// Mitsubishi GX Works2 project: GROUP13   PLC: FX3G

// global labels: Global1
VAR_GLOBAL
  M_StartBlinking AT M100 : BOOL;
  light_generator AT M101 : BOOL;
  TC_BLINK_1 AT TC1 : BOOL;
END_VAR
VAR_GLOBAL CONSTANT
  CONSTANT3_word : INT := 3;
END_VAR
VAR_GLOBAL
  TC_BLINK_2 AT TC2 : BOOL;
  TS_BLINK_1 AT TS1 : BOOL;
  TS_BLINK_2 AT TS2 : BOOL;
  M_BLINKING_LIGHT1 AT M201 : BOOL;
  M_BLINKING_LIGHT2 AT M202 : BOOL;
  Sw_1_Collect AT X001 : BOOL;
  Sw_2_Wash AT X002 : BOOL;
  Sw_3_QA AT X003 : BOOL;
  Sw4 AT X004 : BOOL;
  Sw5 AT X005 : BOOL;
  Sw6 AT X006 : BOOL;
  Sw_7_Emergency AT X007 : BOOL;
  Sw_10_StartDay AT X010 : BOOL;
  Sw_11_Squeeze AT X011 : BOOL;
  Li_1_Collected AT Y001 : BOOL;
  Li_2_Squeeze AT Y002 : BOOL;
  Li_3_Squeeze AT Y003 : BOOL;
  Li_4_QA_Succsed AT Y004 : BOOL;
  Li_5_Wash AT Y005 : BOOL;
  Li6 AT Y006 : BOOL;
  Li7 AT Y007 : BOOL;
  Li_10_Day AT Y010 : BOOL;
  Li11 AT Y011 : BOOL;
  CC_Start_Squeeze_0 AT CC0 : BOOL;
  CS_Start_Squeeze_0 AT CS0 : BOOL;
  TC_Squeeze_10 AT TC10 : BOOL;
END_VAR
VAR_GLOBAL CONSTANT
  CONSTANT2_word : INT := 2;
  CONSTANT30_word : INT := 30;
END_VAR
VAR_GLOBAL
  TS_Squeeze_10 AT TS10 : BOOL;
END_VAR
VAR_GLOBAL CONSTANT
  CONSTANT1_float : REAL := 1;
END_VAR
VAR_GLOBAL
  REG_InvetoryOrange AT D1100 : REAL;
  REG_InvetoryClementine AT D1102 : REAL;
  REG_InvetoryPomelo AT D1104 : REAL;
END_VAR
VAR_GLOBAL CONSTANT
  CONSTANT2_float : REAL := 2;
END_VAR
VAR_GLOBAL
  M_canStartDay AT M0 : BOOL;
  M_TurnOffAll AT M10 : BOOL;
END_VAR
VAR_GLOBAL CONSTANT
  CONSTANT0_float : REAL;
END_VAR
VAR_GLOBAL
  REG_Squeeze AT D1112 : REAL;
  REG_Juice AT D1114 : REAL;
  REG_Storage AT D1116 : REAL;
  TC_CloseDayTimer_3 AT TC3 : BOOL;
  TS_CloseDayTimer_3 AT TS3 : BOOL;
END_VAR
VAR_GLOBAL CONSTANT
  CONSTANT1_word : INT := 1;
END_VAR
VAR_GLOBAL
  M_StartWash AT M1 : BOOL;
  TC_Wash_0 AT TC0 : BOOL;
  TS_Wash_0 AT TS0 : BOOL;
END_VAR
VAR_GLOBAL CONSTANT
  CONSTANT_maxOrange : REAL := 100;
END_VAR
VAR_GLOBAL
  REG_TempWashOrange AT D1118 : REAL;
  M_checkMinimum AT M3 : BOOL;
  REG_minimumPC AT D1120 : REAL;
  M_proportionAdjusment AT M8 : BOOL;
  M_foundMinimum AT M4 : BOOL;
  REG_MinimumPOC AT D1126 : REAL;
  REG_WashOrange AT D1106 : REAL;
  REG_WashClementine AT D1108 : REAL;
  REG_WashPomelo AT D1110 : REAL;
  M_OinWash AT M5 : BOOL;
  M_PinWash AT M6 : BOOL;
  M_CinWash AT M7 : BOOL;
  REG_HalfMinimumPOC AT D1122 : REAL;
  M_Check_QA_1 AT M11 : BOOL;
  M_Check_QA_2 AT M12 : BOOL;
  M_QA_PASSED AT M15 : BOOL;
  M_STARTQA AT M13 : BOOL;
  QA_COUNTER AT CC3 : BOOL;
  CS_MAX_QA AT CS3 : BOOL;
  SW_Analog2_QA AT D8281 : INT;
  REG_QA_value AT D1150 : INT;
END_VAR
VAR_GLOBAL CONSTANT
  CONSTANT5_word : INT := 5;
END_VAR
VAR_GLOBAL
  TC_QA_TEST_PASSED AT TC201 : BOOL;
END_VAR
VAR_GLOBAL CONSTANT
  CONSTANT500_word : INT := 500;
END_VAR
VAR_GLOBAL
  TS_QA_TEST_PASSED AT TS201 : BOOL;
  M_InvetoryOrange_21 AT M21 : BOOL;
  M_InvetoryPomelo_22 AT M22 : BOOL;
  M_InvetoryClementine_20 AT M20 : BOOL;
  M_NotInWash AT M23 : BOOL;
  M_NotInSqueze AT M24 : BOOL;
  M_NotInJuice AT M25 : BOOL;
  REG_keg AT D1128 : INT;
END_VAR
VAR_GLOBAL CONSTANT
  CONSTANT_15_word : INT := 15;
END_VAR
VAR_GLOBAL
  analog_output AT D8282 : INT;
  M_KegNumberFound AT M36 : BOOL;
  REG_keg_FLOAT AT D1132 : REAL;
END_VAR
VAR_GLOBAL CONSTANT
  CONSTANT50_float : REAL := 50;
END_VAR
VAR_GLOBAL
  TS_SHIPMENT_5 AT TS5 : BOOL;
  TC_shipment_5 AT TC5 : BOOL;
  M_SHIMPMENTOVER15 AT M33 : BOOL;
  TC_Shipment_4 AT TC4 : BOOL;
  TS_SHIPMENT_4 AT TS4 : BOOL;
END_VAR
VAR_GLOBAL CONSTANT
  CONSTANT382_1inanalog : INT := 382;
  CONSTANT2020_5inanalog : INT := 2020;
  CONSTANT80_float : REAL := 80;
  CONSTANT_400_word : INT := 400;
END_VAR

// task Task_01 (event TRUE, interval 0, priority 31): POU_01

PROGRAM POU_01
(* structured ladder/FBD written out as ST: instructions are called as NAME(EN, inputs, outputs); _pN, _eN, _tN stand for wires *)
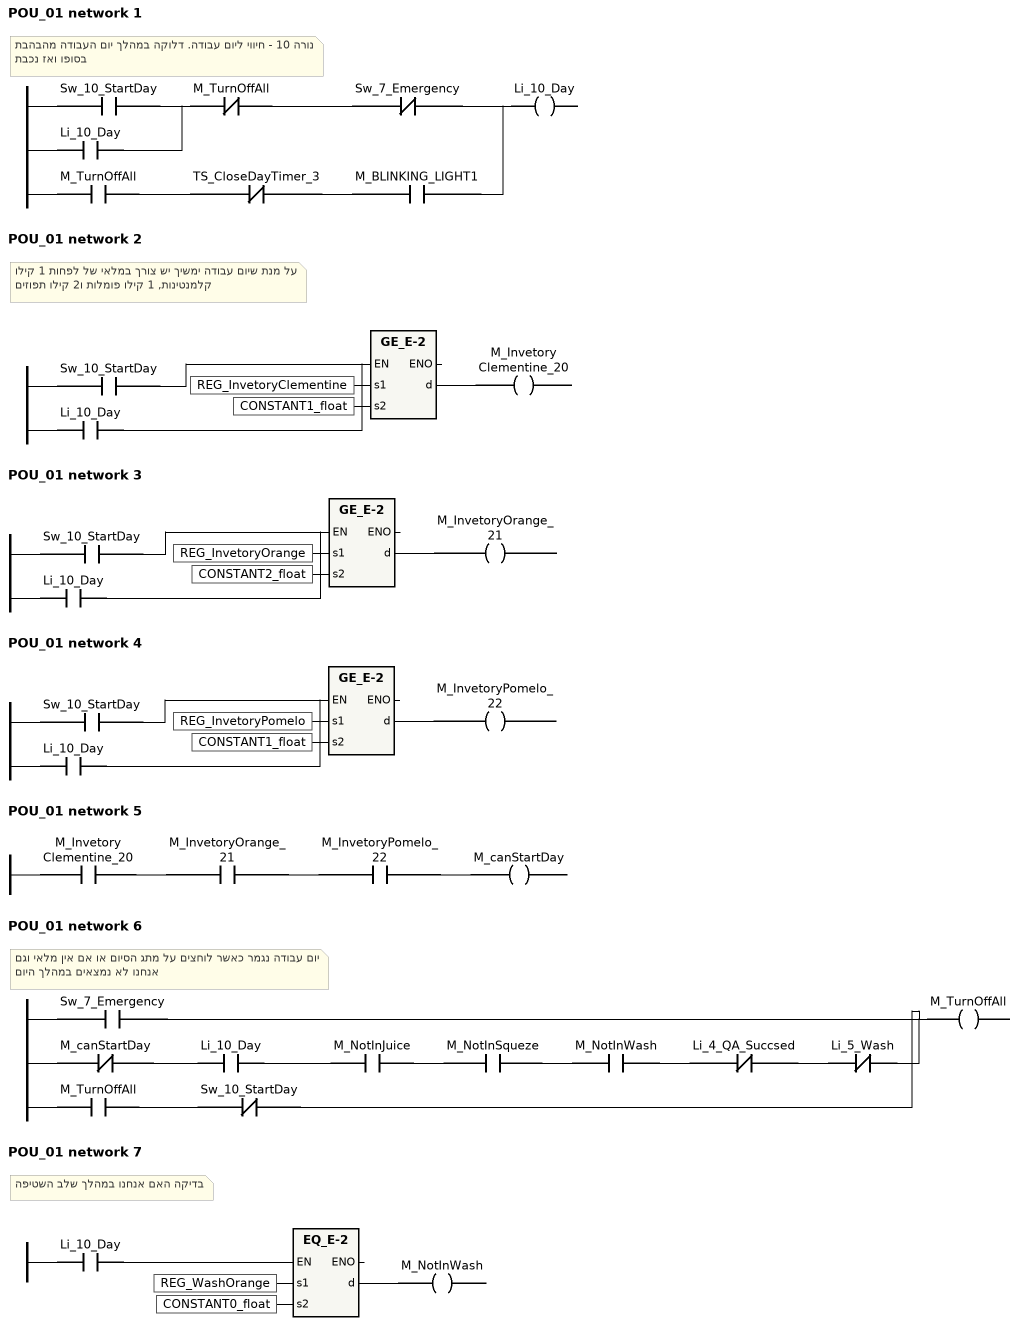
(* network 1 *)
(* נורה 10 - חיווי ליום עבודה. דלוקה במהלך יום העבודה מהבהבת בסופו ואז נכבת *)
Li_10_Day := (((Sw_10_StartDay OR Li_10_Day) AND NOT M_TurnOffAll) AND NOT Sw_7_Emergency) OR (M_TurnOffAll AND NOT TS_CloseDayTimer_3 AND M_BLINKING_LIGHT1);
(* network 2 *)
(* על מנת שיום עבודה ימשיך יש צורך במלאי של לפחות 1 קילו קלמנטינות, 1 קילו פומלות ו2 קילו תפוזים *)
GE_E(Sw_10_StartDay OR Li_10_Day, REG_InvetoryClementine, CONSTANT1_float, _t1);
M_InvetoryClementine_20 := _t1;
(* network 3 *)
GE_E(Sw_10_StartDay OR Li_10_Day, REG_InvetoryOrange, CONSTANT2_float, _t1);
M_InvetoryOrange_21 := _t1;
(* network 4 *)
GE_E(Sw_10_StartDay OR Li_10_Day, REG_InvetoryPomelo, CONSTANT1_float, _t1);
M_InvetoryPomelo_22 := _t1;
(* network 5 *)
M_canStartDay := M_InvetoryClementine_20 AND M_InvetoryOrange_21 AND M_InvetoryPomelo_22;
(* network 6 *)
(* יום עבודה נגמר כאשר לוחצים על מתג הסיום או אם אין מלאי וגם אנחנו לא נמצאים במהלך היום *)
M_TurnOffAll := Sw_7_Emergency OR (NOT M_canStartDay AND Li_10_Day AND M_NotInJuice AND M_NotInSqueze AND M_NotInWash AND NOT Li_4_QA_Succsed AND NOT Li_5_Wash) OR (M_TurnOffAll AND NOT Sw_10_StartDay);
(* network 7 *)
(* בדיקה האם אנחנו במהלך שלב השטיפה *)
EQ_E(Li_10_Day, REG_WashOrange, CONSTANT0_float, _t1);
M_NotInWash := _t1;
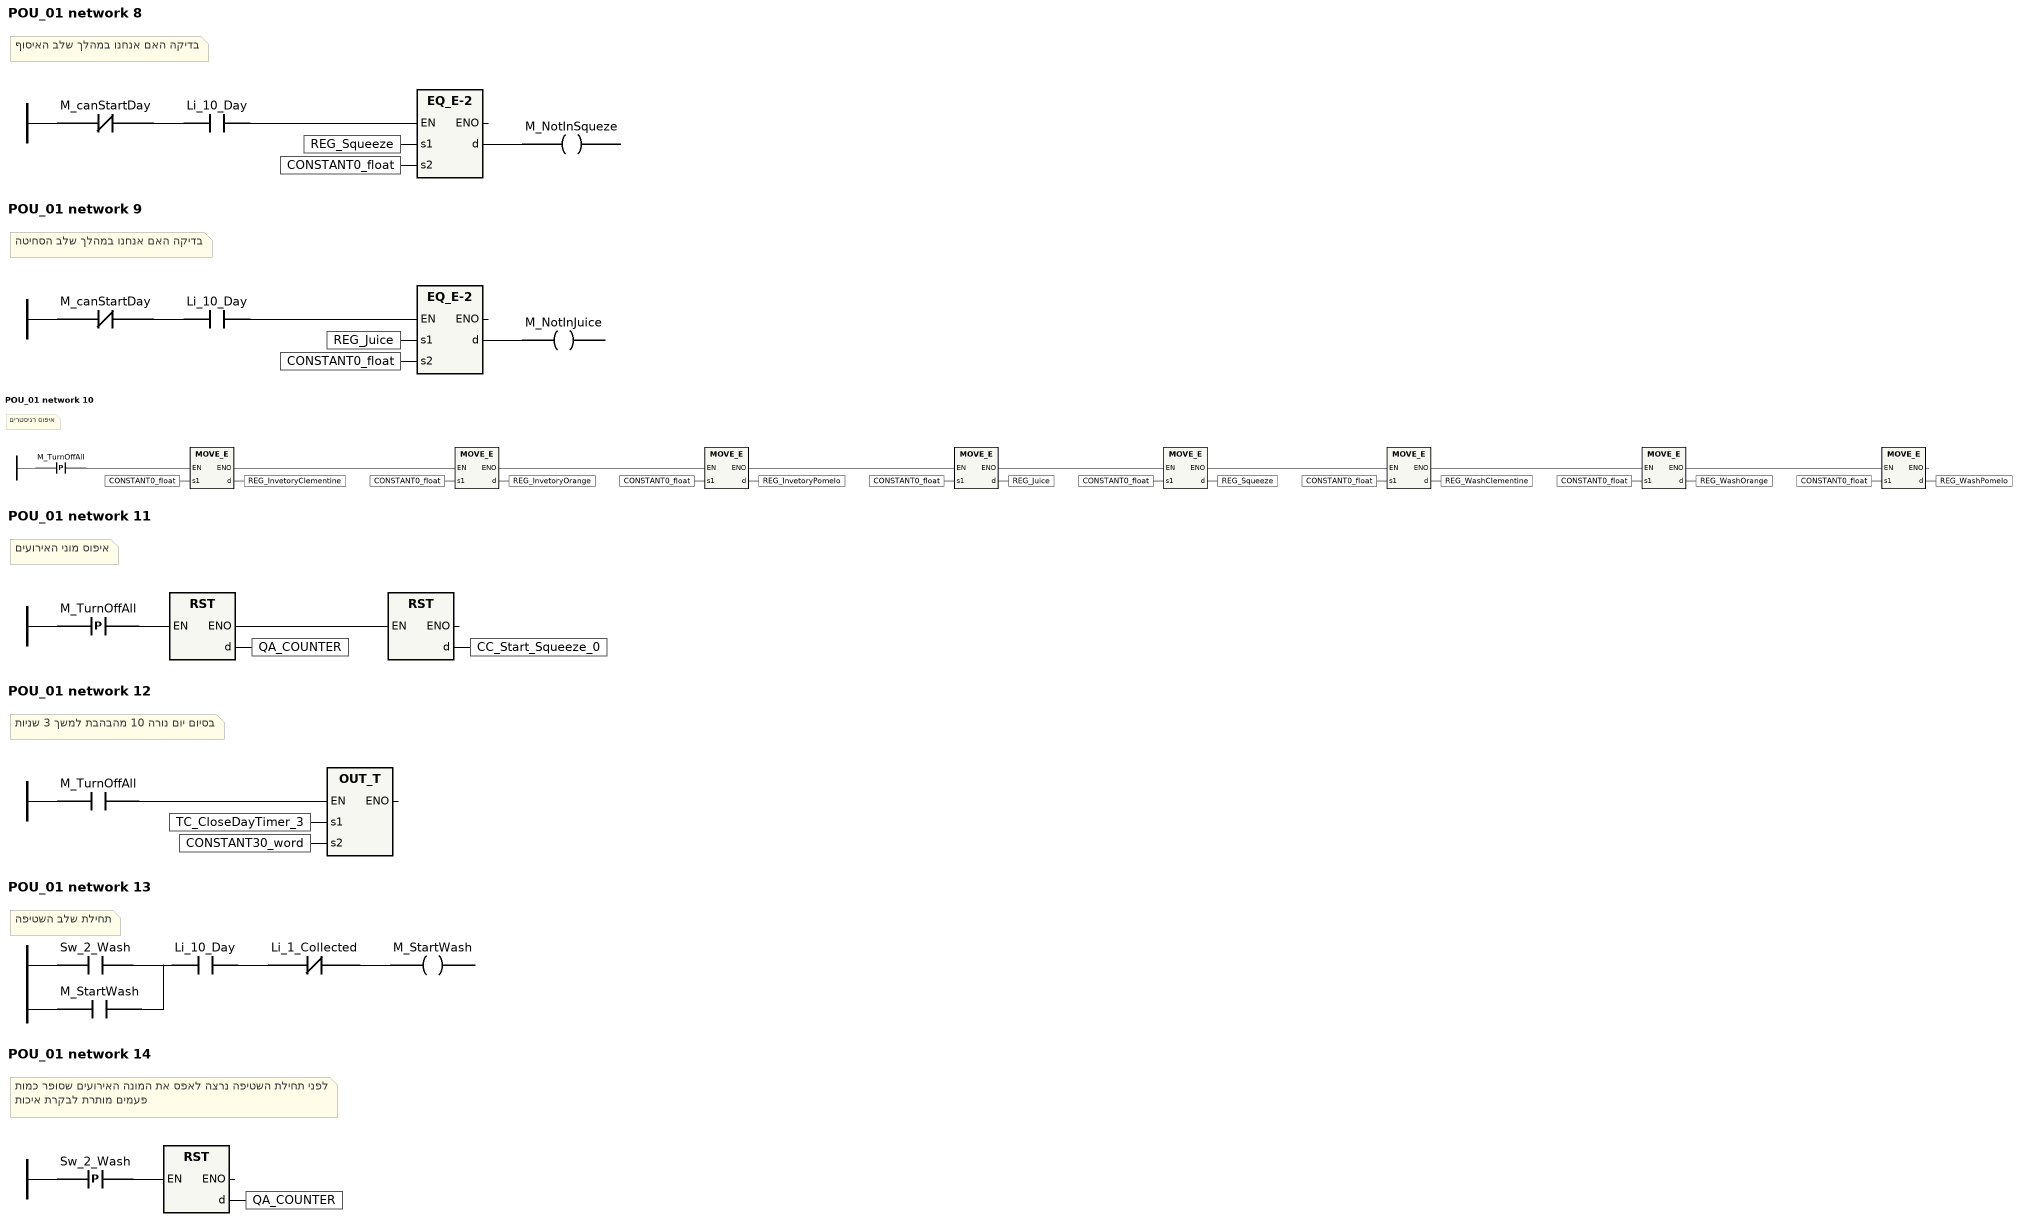
(* network 8 *)
(* בדיקה האם אנחנו במהלך שלב האיסוף *)
EQ_E(NOT M_canStartDay AND Li_10_Day, REG_Squeeze, CONSTANT0_float, _t1);
M_NotInSqueze := _t1;
(* network 9 *)
(* בדיקה האם אנחנו במהלך שלב הסחיטה *)
EQ_E(NOT M_canStartDay AND Li_10_Day, REG_Juice, CONSTANT0_float, _t1);
M_NotInJuice := _t1;
(* network 10 *)
(* איפוס רגיסטרים *)
_e1 := MOVE_E(LDP(TRUE, M_TurnOffAll), CONSTANT0_float, REG_InvetoryClementine);
_e2 := MOVE_E(_e1, CONSTANT0_float, REG_InvetoryOrange);
_e3 := MOVE_E(_e2, CONSTANT0_float, REG_InvetoryPomelo);
_e4 := MOVE_E(_e3, CONSTANT0_float, REG_Juice);
_e5 := MOVE_E(_e4, CONSTANT0_float, REG_Squeeze);
_e6 := MOVE_E(_e5, CONSTANT0_float, REG_WashClementine);
_e7 := MOVE_E(_e6, CONSTANT0_float, REG_WashOrange);
MOVE_E(_e7, CONSTANT0_float, REG_WashPomelo);
(* network 11 *)
(* איפוס מוני האירועים *)
_e1 := RST(LDP(TRUE, M_TurnOffAll), QA_COUNTER);
RST(_e1, CC_Start_Squeeze_0);
(* network 12 *)
(* בסיום יום נורה 10 מהבהבת למשך 3 שניות *)
OUT_T(M_TurnOffAll, TC_CloseDayTimer_3, CONSTANT30_word);
(* network 13 *)
(* תחילת שלב השטיפה *)
M_StartWash := ((Sw_2_Wash OR M_StartWash) AND Li_10_Day) AND NOT Li_1_Collected;
(* network 14 *)
(* לפני תחילת השטיפה נרצה לאפס את המונה האירועים שסופר כמות פעמים מותרת לבקרת איכות *)
RST(LDP(TRUE, Sw_2_Wash), QA_COUNTER);
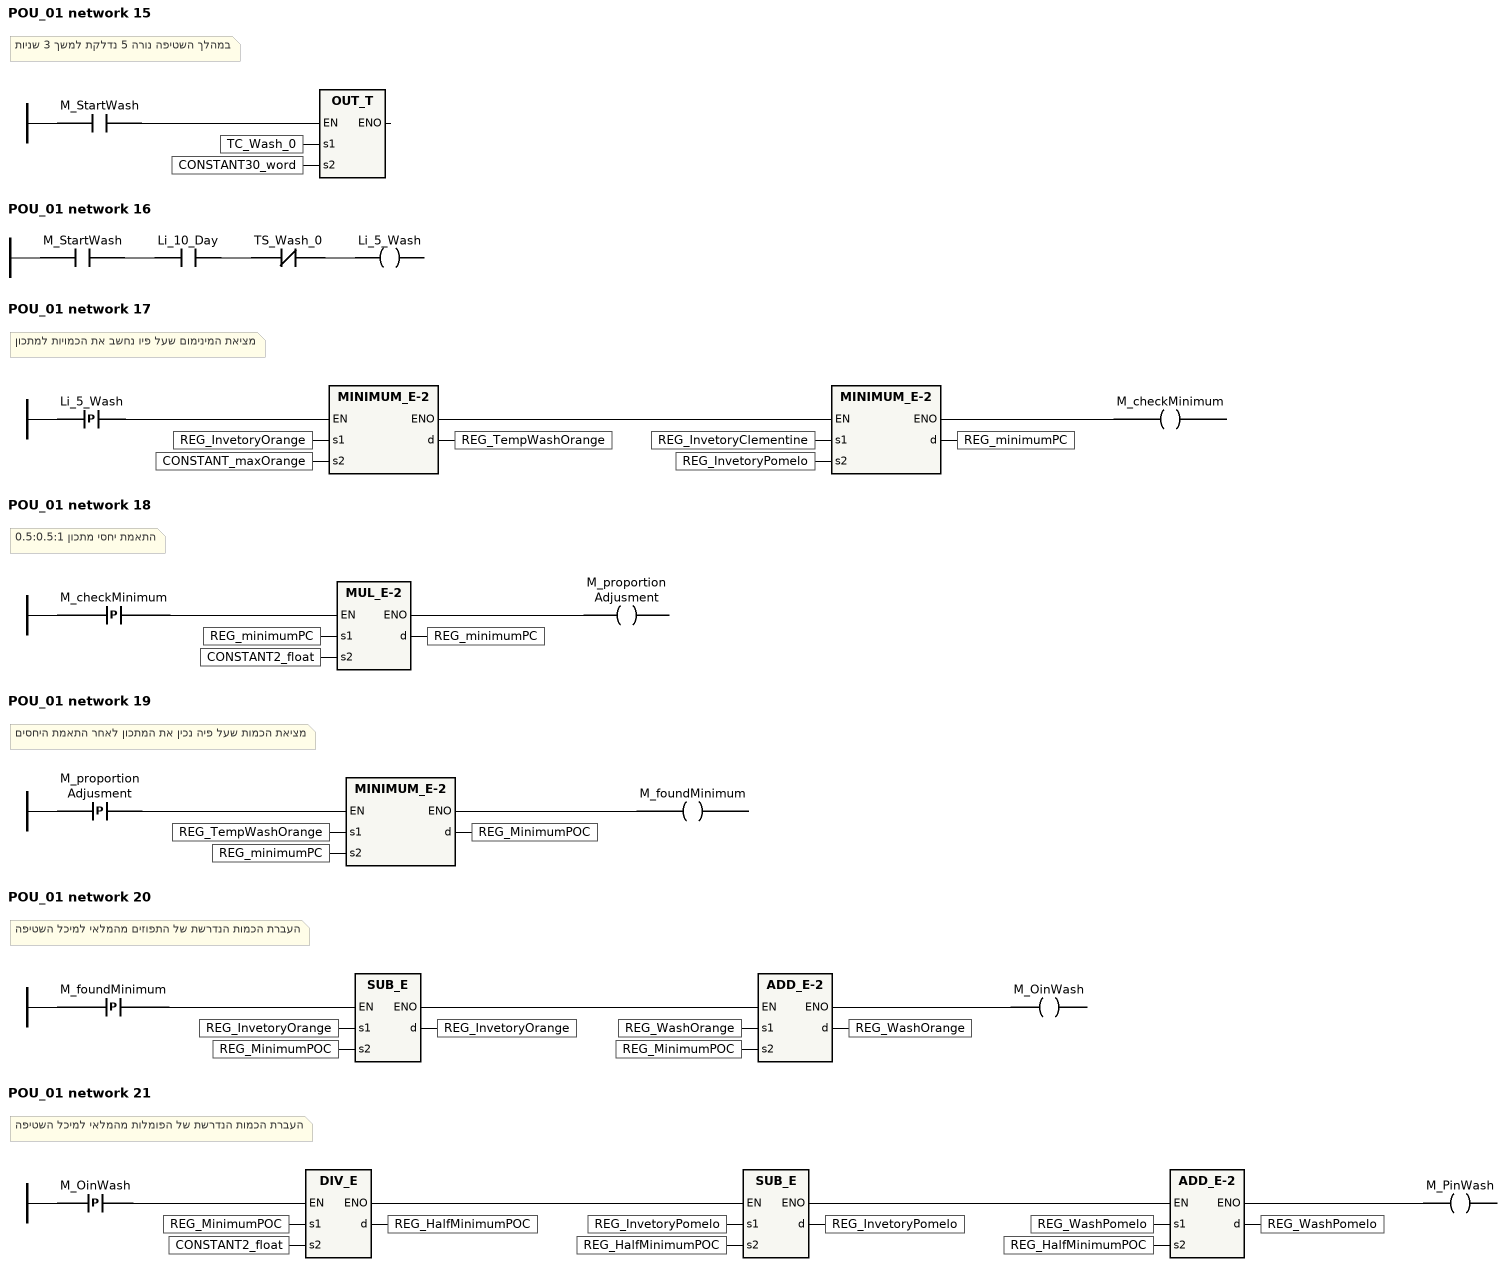
(* network 15 *)
(* במהלך השטיפה נורה 5 נדלקת למשך 3 שניות *)
OUT_T(M_StartWash, TC_Wash_0, CONSTANT30_word);
(* network 16 *)
Li_5_Wash := M_StartWash AND Li_10_Day AND NOT TS_Wash_0;
(* network 17 *)
(* מציאת המינימום שעל פיו נחשב את הכמויות למתכון *)
_e1 := MINIMUM_E(LDP(TRUE, Li_5_Wash), REG_InvetoryOrange, CONSTANT_maxOrange, REG_TempWashOrange);
_e2 := MINIMUM_E(_e1, REG_InvetoryClementine, REG_InvetoryPomelo, REG_minimumPC);
M_checkMinimum := _e2;
(* network 18 *)
(* התאמת יחסי מתכון 0.5:0.5:1 *)
_e1 := MUL_E(LDP(TRUE, M_checkMinimum), REG_minimumPC, CONSTANT2_float, REG_minimumPC);
M_proportionAdjusment := _e1;
(* network 19 *)
(* מציאת הכמות שעל פיה נכין את המתכון לאחר התאמת היחסים *)
_e1 := MINIMUM_E(LDP(TRUE, M_proportionAdjusment), REG_TempWashOrange, REG_minimumPC, REG_MinimumPOC);
M_foundMinimum := _e1;
(* network 20 *)
(* העברת הכמות הנדרשת של התפוזים מהמלאי למיכל השטיפה *)
_e1 := SUB_E(LDP(TRUE, M_foundMinimum), REG_InvetoryOrange, REG_MinimumPOC, REG_InvetoryOrange);
_e2 := ADD_E(_e1, REG_WashOrange, REG_MinimumPOC, REG_WashOrange);
M_OinWash := _e2;
(* network 21 *)
(* העברת הכמות הנדרשת של הפומלות מהמלאי למיכל השטיפה *)
_e1 := DIV_E(LDP(TRUE, M_OinWash), REG_MinimumPOC, CONSTANT2_float, REG_HalfMinimumPOC);
_e2 := SUB_E(_e1, REG_InvetoryPomelo, REG_HalfMinimumPOC, REG_InvetoryPomelo);
_e3 := ADD_E(_e2, REG_WashPomelo, REG_HalfMinimumPOC, REG_WashPomelo);
M_PinWash := _e3;
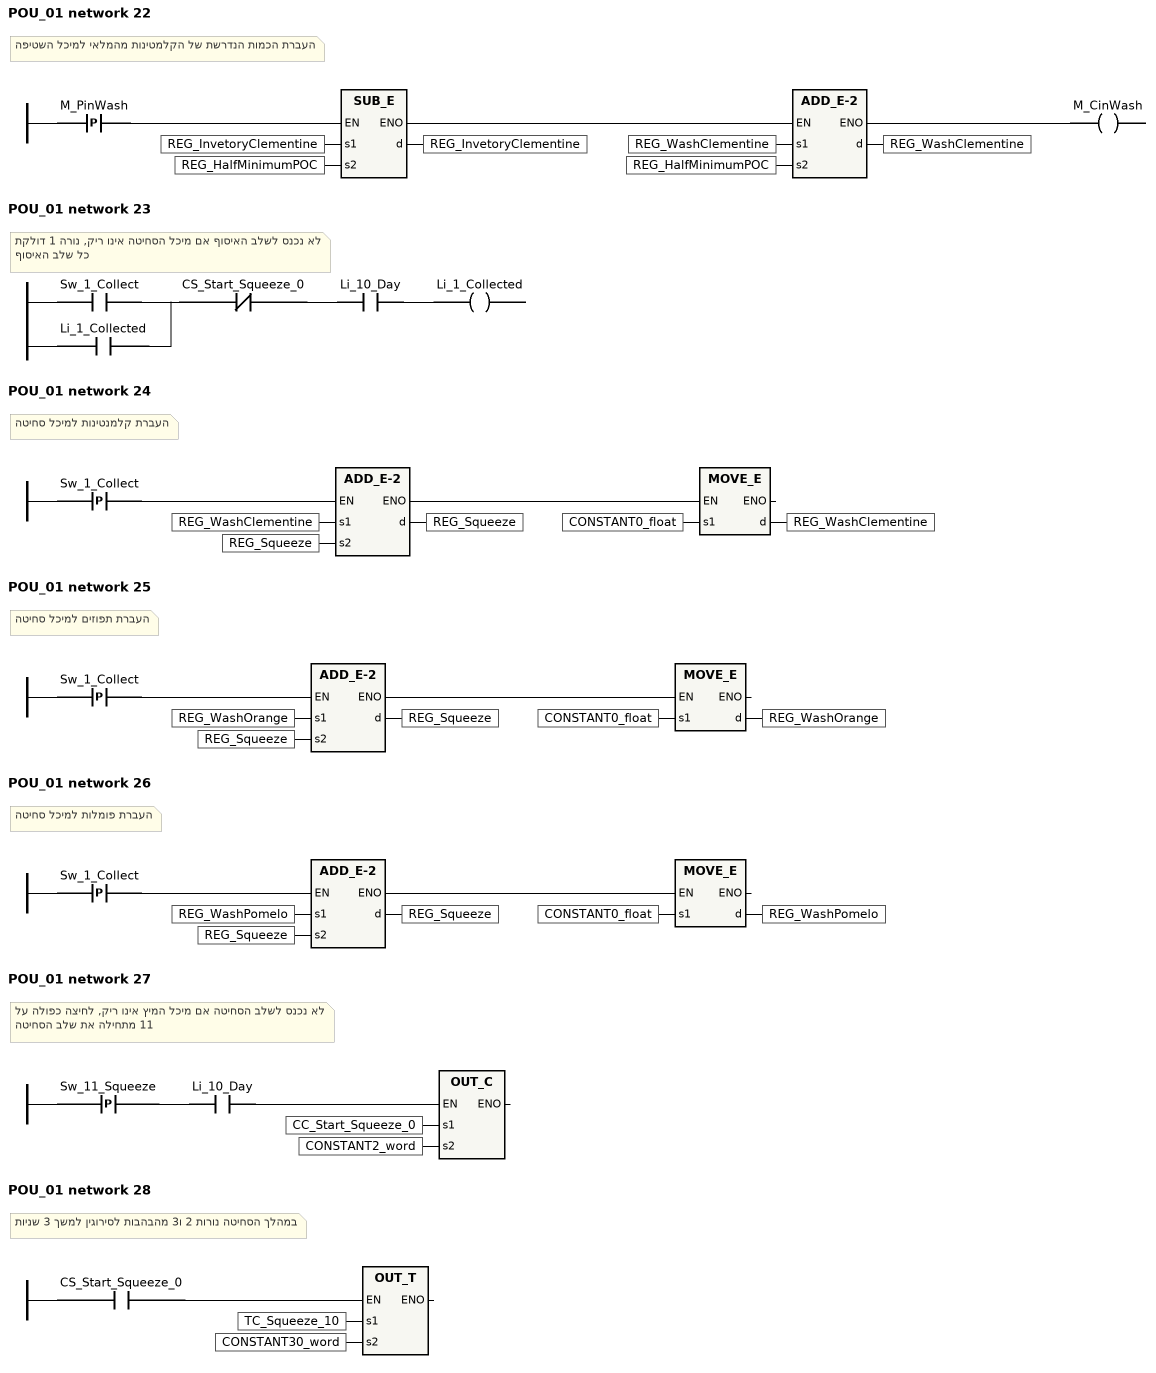
(* network 22 *)
(* העברת הכמות הנדרשת של הקלמטינות מהמלאי למיכל השטיפה *)
_e1 := SUB_E(LDP(TRUE, M_PinWash), REG_InvetoryClementine, REG_HalfMinimumPOC, REG_InvetoryClementine);
_e2 := ADD_E(_e1, REG_WashClementine, REG_HalfMinimumPOC, REG_WashClementine);
M_CinWash := _e2;
(* network 23 *)
(* לא נכנס לשלב האיסוף אם מיכל הסחיטה אינו ריק, נורה 1 דולקת כל שלב האיסוף *)
Li_1_Collected := ((Sw_1_Collect OR Li_1_Collected) AND NOT CS_Start_Squeeze_0) AND Li_10_Day;
(* network 24 *)
(* העברת קלמנטינות למיכל סחיטה *)
_e1 := ADD_E(LDP(TRUE, Sw_1_Collect), REG_WashClementine, REG_Squeeze, REG_Squeeze);
MOVE_E(_e1, CONSTANT0_float, REG_WashClementine);
(* network 25 *)
(* העברת תפוזים למיכל סחיטה *)
_e1 := ADD_E(LDP(TRUE, Sw_1_Collect), REG_WashOrange, REG_Squeeze, REG_Squeeze);
MOVE_E(_e1, CONSTANT0_float, REG_WashOrange);
(* network 26 *)
(* העברת פומלות למיכל סחיטה *)
_e1 := ADD_E(LDP(TRUE, Sw_1_Collect), REG_WashPomelo, REG_Squeeze, REG_Squeeze);
MOVE_E(_e1, CONSTANT0_float, REG_WashPomelo);
(* network 27 *)
(* לא נכנס לשלב הסחיטה אם מיכל המיץ אינו ריק, לחיצה כפולה על 11 מתחילה את שלב הסחיטה *)
OUT_C(LDP(TRUE, Sw_11_Squeeze) AND Li_10_Day, CC_Start_Squeeze_0, CONSTANT2_word);
(* network 28 *)
(* במהלך הסחיטה נורות 2 ו3 מהבהבות לסירוגין למשך 3 שניות *)
OUT_T(CS_Start_Squeeze_0, TC_Squeeze_10, CONSTANT30_word);
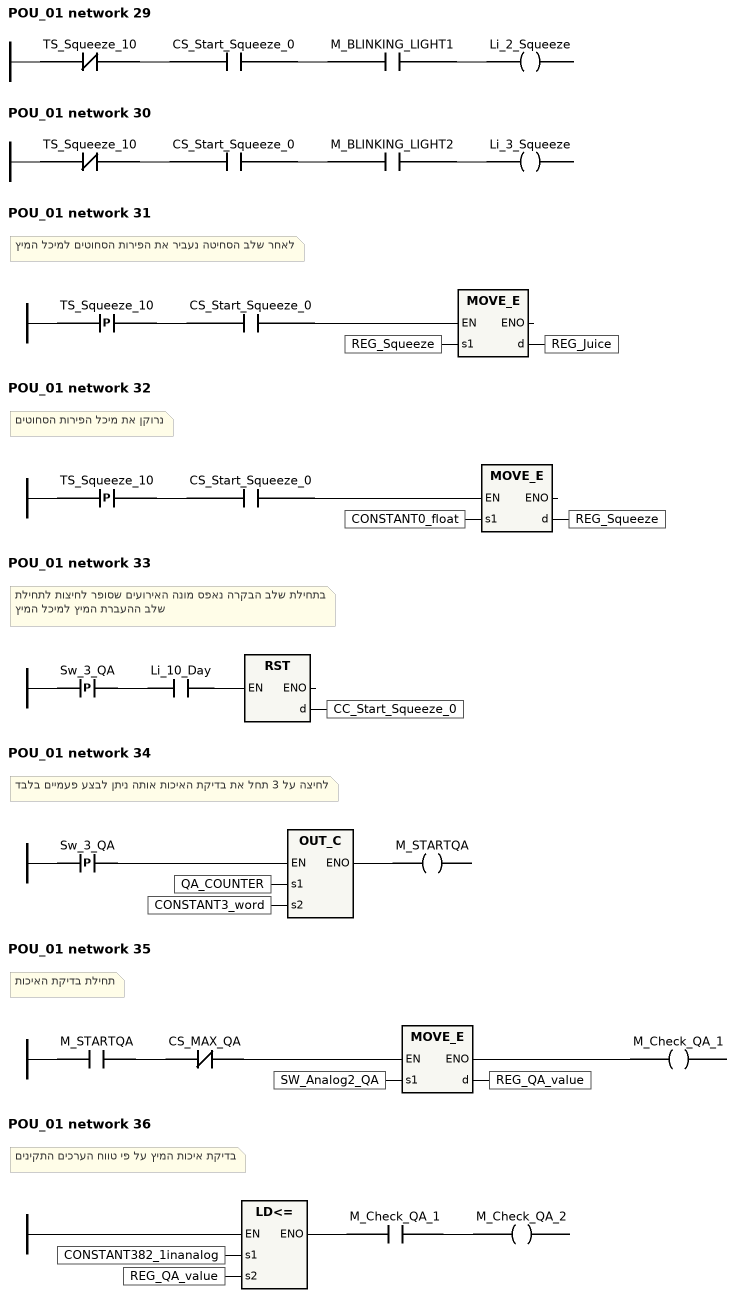
(* network 29 *)
Li_2_Squeeze := NOT TS_Squeeze_10 AND CS_Start_Squeeze_0 AND M_BLINKING_LIGHT1;
(* network 30 *)
Li_3_Squeeze := NOT TS_Squeeze_10 AND CS_Start_Squeeze_0 AND M_BLINKING_LIGHT2;
(* network 31 *)
(* לאחר שלב הסחיטה נעביר את הפירות הסחוטים למיכל המיץ *)
MOVE_E(LDP(TRUE, TS_Squeeze_10) AND CS_Start_Squeeze_0, REG_Squeeze, REG_Juice);
(* network 32 *)
(* נרוקן את מיכל הפירות הסחוטים *)
MOVE_E(LDP(TRUE, TS_Squeeze_10) AND CS_Start_Squeeze_0, CONSTANT0_float, REG_Squeeze);
(* network 33 *)
(* בתחילת שלב הבקרה נאפס מונה האירועים שסופר לחיצות לתחילת שלב ההעברת המיץ למיכל המיץ *)
RST(LDP(TRUE, Sw_3_QA) AND Li_10_Day, CC_Start_Squeeze_0);
(* network 34 *)
(* לחיצה על 3 תחל את בדיקת האיכות אותה ניתן לבצע פעמיים בלבד *)
_e1 := OUT_C(LDP(TRUE, Sw_3_QA), QA_COUNTER, CONSTANT3_word);
M_STARTQA := _e1;
(* network 35 *)
(* תחילת בדיקת האיכות *)
_e1 := MOVE_E(M_STARTQA AND NOT CS_MAX_QA, SW_Analog2_QA, REG_QA_value);
M_Check_QA_1 := _e1;
(* network 36 *)
(* בדיקת איכות המיץ על פי טווח הערכים התקינים *)
_e1 := LD<=(TRUE, CONSTANT382_1inanalog, REG_QA_value);
M_Check_QA_2 := _e1 AND M_Check_QA_1;
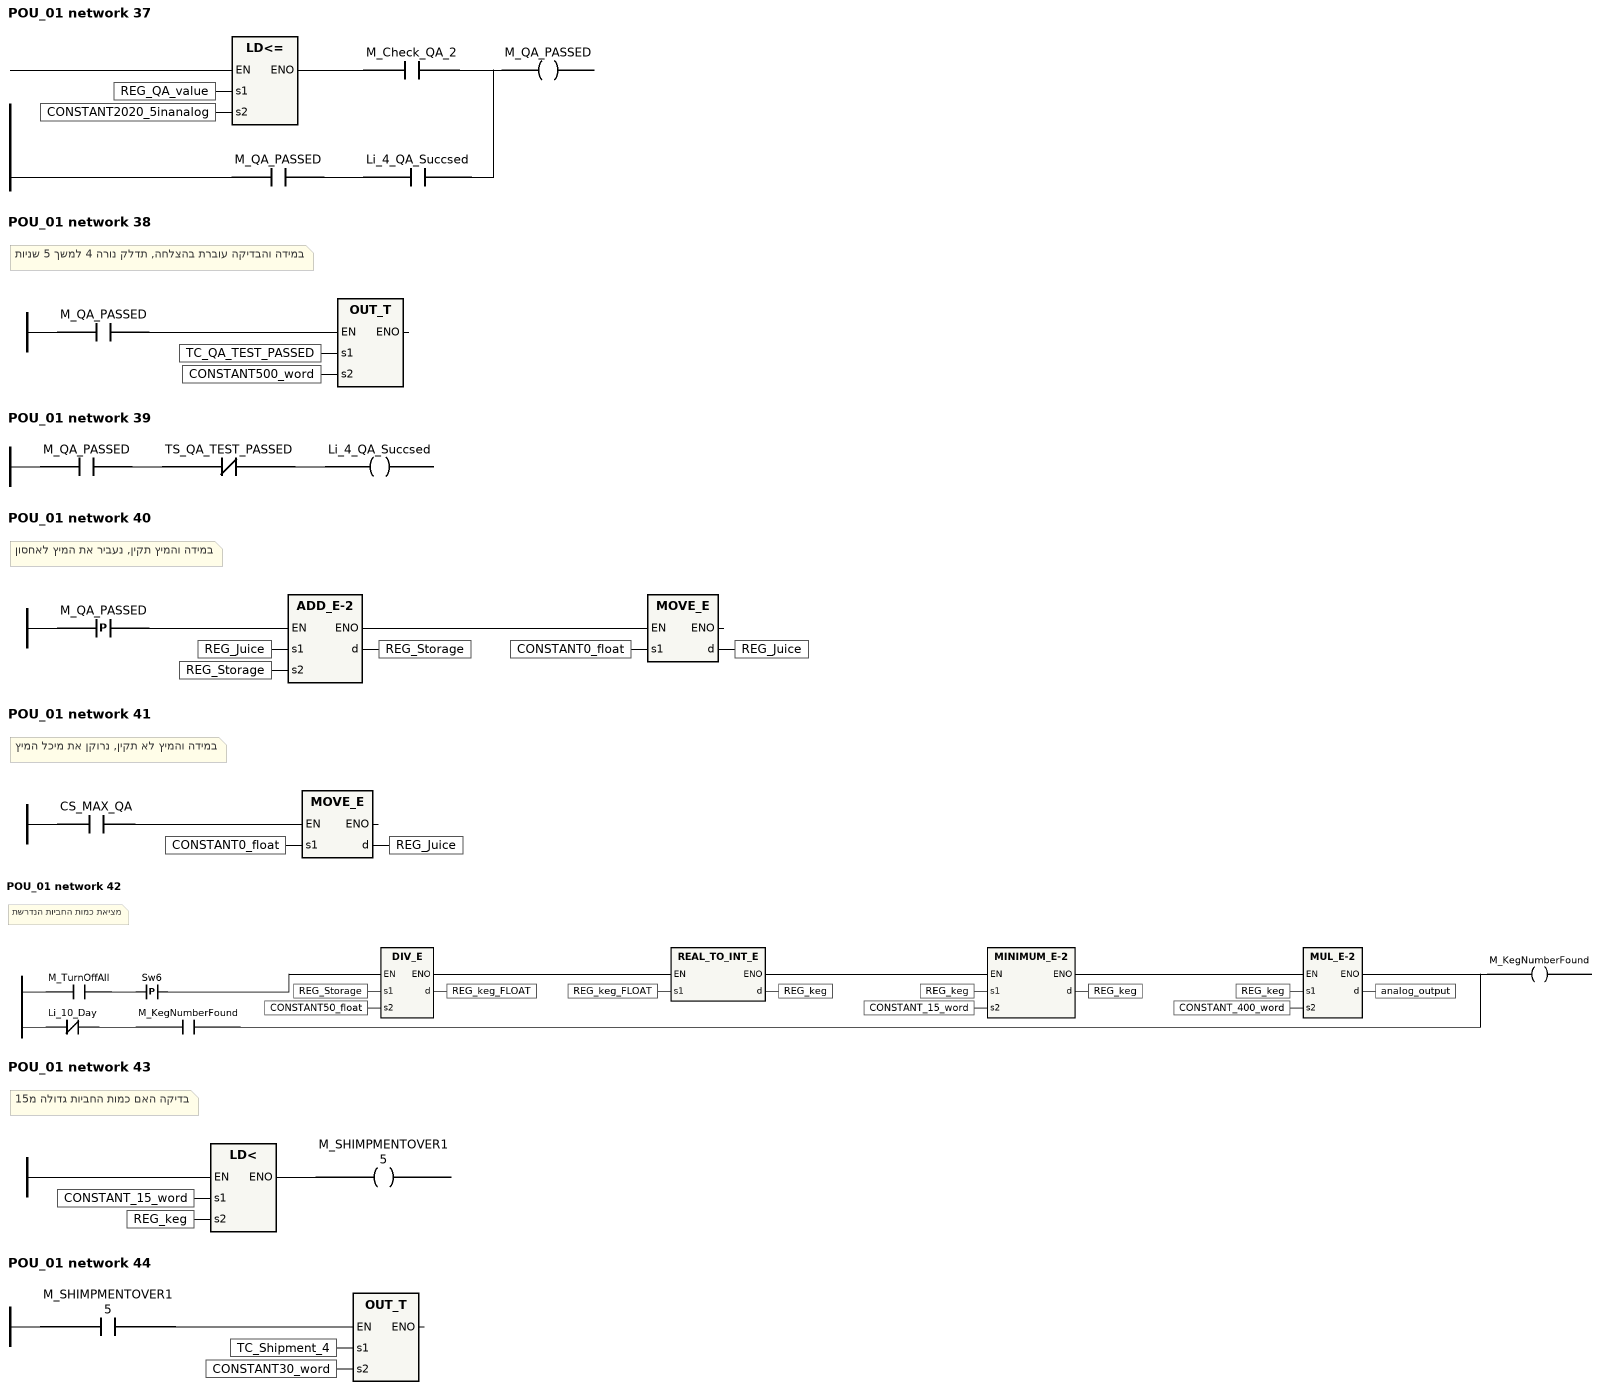
(* network 37 *)
_e1 := LD<=(TRUE, REG_QA_value, CONSTANT2020_5inanalog);
M_QA_PASSED := (_e1 AND M_Check_QA_2) OR (M_QA_PASSED AND Li_4_QA_Succsed);
(* network 38 *)
(* במידה והבדיקה עוברת בהצלחה, תדלק נורה 4 למשך 5 שניות *)
OUT_T(M_QA_PASSED, TC_QA_TEST_PASSED, CONSTANT500_word);
(* network 39 *)
Li_4_QA_Succsed := M_QA_PASSED AND NOT TS_QA_TEST_PASSED;
(* network 40 *)
(* במידה והמיץ תקין, נעביר את המיץ לאחסון *)
_e1 := ADD_E(LDP(TRUE, M_QA_PASSED), REG_Juice, REG_Storage, REG_Storage);
MOVE_E(_e1, CONSTANT0_float, REG_Juice);
(* network 41 *)
(* במידה והמיץ לא תקין, נרוקן את מיכל המיץ *)
MOVE_E(CS_MAX_QA, CONSTANT0_float, REG_Juice);
(* network 42 *)
(* מציאת כמות החביות הנדרשת *)
_e1 := DIV_E(M_TurnOffAll AND LDP(TRUE, Sw6), REG_Storage, CONSTANT50_float, REG_keg_FLOAT);
_e2 := REAL_TO_INT_E(_e1, REG_keg_FLOAT, REG_keg);
_e3 := MINIMUM_E(_e2, REG_keg, CONSTANT_15_word, REG_keg);
_e4 := MUL_E(_e3, REG_keg, CONSTANT_400_word, analog_output);
M_KegNumberFound := _e4 OR (NOT Li_10_Day AND M_KegNumberFound);
(* network 43 *)
(* בדיקה האם כמות החביות גדולה מ15 *)
_e1 := LD<(TRUE, CONSTANT_15_word, REG_keg);
M_SHIMPMENTOVER15 := _e1;
(* network 44 *)
OUT_T(M_SHIMPMENTOVER15, TC_Shipment_4, CONSTANT30_word);
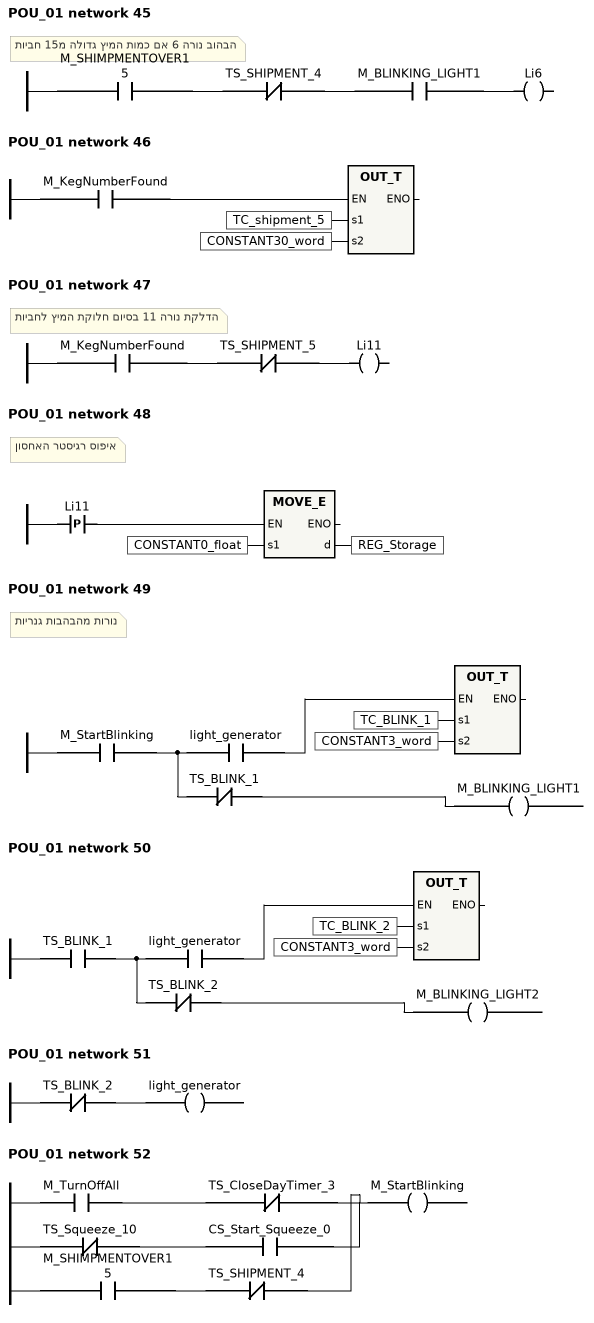
(* network 45 *)
(* הבהוב נורה 6 אם כמות המיץ גדולה מ15 חביות *)
Li6 := M_SHIMPMENTOVER15 AND NOT TS_SHIPMENT_4 AND M_BLINKING_LIGHT1;
(* network 46 *)
OUT_T(M_KegNumberFound, TC_shipment_5, CONSTANT30_word);
(* network 47 *)
(* הדלקת נורה 11 בסיום חלוקת המיץ לחביות *)
Li11 := M_KegNumberFound AND NOT TS_SHIPMENT_5;
(* network 48 *)
(* איפוס רגיסטר האחסון *)
MOVE_E(LDP(TRUE, Li11), CONSTANT0_float, REG_Storage);
(* network 49 *)
(* נורות מהבהבות גנריות *)
OUT_T(M_StartBlinking AND light_generator, TC_BLINK_1, CONSTANT3_word);
M_BLINKING_LIGHT1 := M_StartBlinking AND NOT TS_BLINK_1;
(* network 50 *)
OUT_T(TS_BLINK_1 AND light_generator, TC_BLINK_2, CONSTANT3_word);
M_BLINKING_LIGHT2 := TS_BLINK_1 AND NOT TS_BLINK_2;
(* network 51 *)
light_generator := NOT TS_BLINK_2;
(* network 52 *)
M_StartBlinking := (M_TurnOffAll AND NOT TS_CloseDayTimer_3) OR (NOT TS_Squeeze_10 AND CS_Start_Squeeze_0) OR (M_SHIMPMENTOVER15 AND NOT TS_SHIPMENT_4);
END_PROGRAM
